Fanuc KAREL source: RUN_TASK.kl

PROGRAM T
%NOLOCKGROUP
VAR
 v0 : STRING[40]
 v1 : INTEGER
 v2 : BOOLEAN
 v3 : BOOLEAN
 v4 : INTEGER
 v5 : INTEGER
BEGIN
 RUN_TASK(v0, v1, v2, v3, v4, v5)
END T
